// TIA Portal V20 export
DATA_BLOCK "UnitModule_DB"   // DB1
// stored: AssignedProDiagFB ProDiag, InstanceOfName UnitModule, InstanceOfType FB
"UnitModule"
   // VAR
   //    IOInterface : "IOInterface";
   //    CMInterface { ExternalAccessible := 'False'; ExternalVisible := 'False'; ExternalWritable := 'False'} : "CMInterface";
   //    CM : "CMs";
   //    Sim { ExternalAccessible := 'False'; ExternalVisible := 'False'; ExternalWritable := 'False'} : "Simulate";
   //    Inputs { ExternalAccessible := 'False'; ExternalVisible := 'False'; ExternalWritable := 'False'} : "MapInputs";
   //    Outputs { ExternalAccessible := 'False'; ExternalVisible := 'False'; ExternalWritable := 'False'} : "MapOutputs";
   //    Simulate { ExternalAccessible := 'False'; ExternalVisible := 'False'; ExternalWritable := 'False'} : Bool;
   // END_VAR
BEGIN
END_DATA_BLOCK
